PROGRAM DNS_REV_DEMO
VAR
	DNS_REV_CLIENT: DNS_REV_CLIENT;
	IP_C : IP_C;
	S_BUF : NETWORK_BUFFER;
	R_BUF : NETWORK_BUFFER;
	IP_CONTROL : IP_CONTROL;
	activate : BOOL := TRUE;
	done : BOOL;
	error: DWORD;
	domain: STRING;
END_VAR
VAR // added by the converter: edge detectors and wires of the graphical bodies
    _w1, _w2 : ANY;
END_VAR

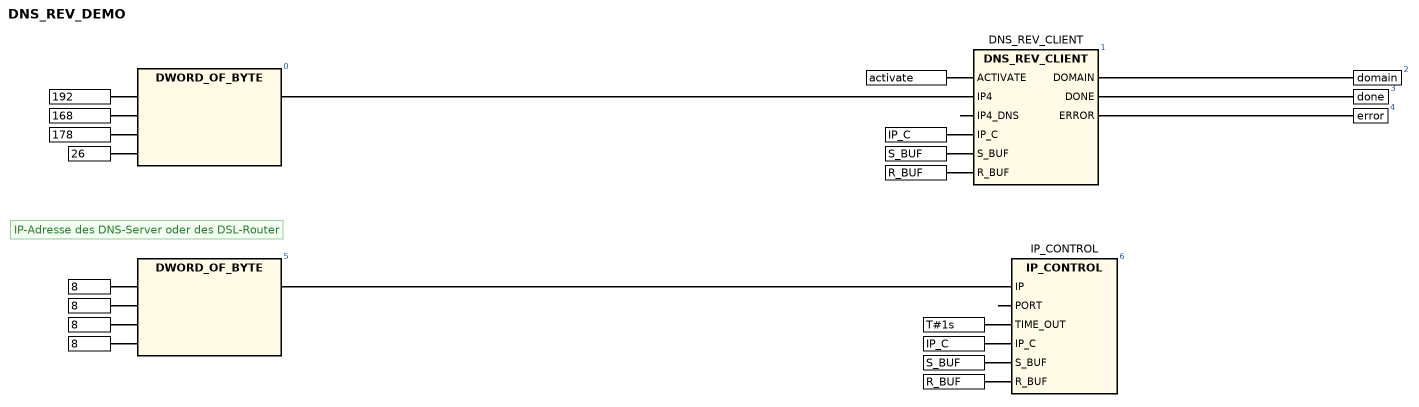
_w1 := DWORD_OF_BYTE(192, 168, 178, 26);
DNS_REV_CLIENT(ACTIVATE := activate, IP4 := _w1, IP_C := IP_C, S_BUF := S_BUF, R_BUF := R_BUF);
domain := DNS_REV_CLIENT.DOMAIN;
done := DNS_REV_CLIENT.DONE;
error := DNS_REV_CLIENT.ERROR;
// IP-Adresse des DNS-Server oder des DSL-Router
_w2 := DWORD_OF_BYTE(8, 8, 8, 8);
IP_CONTROL(IP := _w2, TIME_OUT := T#1s, IP_C := IP_C, S_BUF := S_BUF, R_BUF := R_BUF);

END_PROGRAM

(* stored: Version 1.1.0.1, ProductVersion 3.1.4024.9
   POU DNS_REV_DEMO: Id {943c9808-d3a1-4ef5-b5e1-aa16ccac4da6}, SpecialFunc None *)
